// TIA Portal V20 export
DATA_BLOCK "Instance_FB_Digital_Outputs_DB"   // DB103
// stored: AutoNumber false, InstanceOfName FB_Digital_Outputs, InstanceOfType FB
"FB_Digital_Outputs"
   // VAR_INPUT
   //    DB_Digital_Output_0 : Bool;
   //    DB_Digital_Output_1 : Bool;
   //    DB_Digital_Output_2 : Bool;
   //    DB_Digital_Output_3 : Bool;
   //    DB_Digital_Output_4 : Bool;
   //    DB_Digital_Output_5 : Bool;
   //    DB_Digital_Output_6 : Bool;
   //    DB_Digital_Output_7 : Bool;
   //    DB_Digital_Output_8 : Bool;
   //    DB_Digital_Output_9 : Bool;
   // END_VAR
   // VAR_OUTPUT
   //    Q_Digital_Output_0 : Bool;
   //    Q_Digital_Output_1 : Bool;
   //    Q_Digital_Output_2 : Bool;
   //    Q_Digital_Output_3 : Bool;
   //    Q_Digital_Output_4 : Bool;
   //    Q_Digital_Output_5 : Bool;
   //    Q_Digital_Output_6 : Bool;
   //    Q_Digital_Output_7 : Bool;
   //    Q_Digital_Output_8 : Bool;
   //    Q_Digital_Output_9 : Bool;
   // END_VAR
BEGIN
END_DATA_BLOCK
